{attribute 'GeneratedUsingTerminal: EL6752--0000'}
{attribute addProperty BoxType "EL6752--0000"}
{attribute addProperty Id "InfoDataAT %I*InfoData_41C547A32"}
{attribute addProperty CRC "3204926373"}
{attribute addProperty Size "2"}
TYPE EL6752_BF074BA5 EXTENDS EtcSlaveTerminalBase_947E5A46 :
STRUCT
	{attribute addProperty Name "InfoData"}
	InfoData : InfoData_41C547A3;
END_STRUCT
END_TYPE

(* stored: Version 1.2.0.0, ProductVersion 3.1.4024.9
   DUT EL6752_BF074BA5: Id {2e4cb495-cef3-46aa-8985-d3c01d0a569f} *)
